PROGRAM PRG_Test
VAR
	fbBaseTimeTest			: FB_BaseTimeTest;

	fbBaseTest				: FB_Basetest;
	fbComponentTest			: FB_ElementTest;
END_VAR


	TcUnit.RUN_IN_SEQUENCE ();

END_PROGRAM

(* stored: Version 1.1.0.1, ProductVersion 3.1.4024.15
   POU PRG_Test: Id {08f2cb9f-fc15-489b-a378-35435c110658}, SpecialFunc None *)
